LIN {X 121.514,Y -7.144,Z -55.406,A -90.000,B 90.000,C 0.000} C_DIS
LIN {X 120.744,Y -7.144,Z -56.976,A -90.000,B 90.000,C 0.000} C_DIS
LIN {X 120.185,Y -7.144,Z -58.438,A -90.000,B 90.000,C 0.000} C_DIS
LIN {X 119.652,Y -7.144,Z -59.909,A -90.000,B 90.000,C 0.000} C_DIS
LIN {X 119.147,Y -7.144,Z -61.390,A -90.000,B 90.000,C 0.000} C_DIS
LIN {X 144.015,Y -7.144,Z -61.390,A -90.000,B 90.000,C 0.000} C_DIS
LIN {X 144.015,Y -7.144,Z -68.939,A -90.000,B 90.000,C 0.000} C_DIS
LIN {X 116.917,Y -7.144,Z -68.939,A -90.000,B 90.000,C 0.000} C_DIS
LIN {X 116.287,Y -7.144,Z -70.857,A -90.000,B 90.000,C 0.000} C_DIS
LIN {X 115.601,Y -7.144,Z -72.756,A -90.000,B 90.000,C 0.000} C_DIS
LIN {X 114.859,Y -7.144,Z -74.633,A -90.000,B 90.000,C 0.000} C_DIS
LIN {X 114.062,Y -7.144,Z -76.488,A -90.000,B 90.000,C 0.000} C_DIS
LIN {X 144.015,Y -7.144,Z -76.488,A -90.000,B 90.000,C 0.000} C_DIS
LIN {X 144.015,Y -7.144,Z -84.037,A -90.000,B 90.000,C 0.000} C_DIS
LIN {X 110.374,Y -7.144,Z -84.037,A -90.000,B 90.000,C 0.000} C_DIS
LIN {X 110.982,Y -7.144,Z -85.267,A -90.000,B 90.000,C 0.000} C_DIS
LIN {X 111.542,Y -7.144,Z -86.519,A -90.000,B 90.000,C 0.000} C_DIS
LIN {X 112.054,Y -7.144,Z -87.792,A -90.000,B 90.000,C 0.000} C_DIS
LIN {X 112.517,Y -7.144,Z -89.084,A -90.000,B 90.000,C 0.000} C_DIS
LIN {X 112.888,Y -7.144,Z -90.333,A -90.000,B 90.000,C 0.000} C_DIS
LIN {X 113.248,Y -7.144,Z -91.586,A -90.000,B 90.000,C 0.000} C_DIS
LIN {X 144.015,Y -7.144,Z -91.586,A -90.000,B 90.000,C 0.000} C_DIS
LIN {X 144.015,Y -7.144,Z -99.134,A -90.000,B 90.000,C 0.000} C_DIS
LIN {X 115.197,Y -7.144,Z -99.134,A -90.000,B 90.000,C 0.000} C_DIS
LIN {X 115.413,Y -7.144,Z -100.073,A -90.000,B 90.000,C 0.000} C_DIS
LIN {X 115.939,Y -7.144,Z -102.270,A -90.000,B 90.000,C 0.000} C_DIS
LIN {X 116.438,Y -7.144,Z -104.473,A -90.000,B 90.000,C 0.000} C_DIS
LIN {X 116.908,Y -7.144,Z -106.683,A -90.000,B 90.000,C 0.000} C_DIS
LIN {X 144.015,Y -7.144,Z -106.683,A -90.000,B 90.000,C 0.000} C_DIS
LIN {X 144.015,Y -7.144,Z -114.232,A -90.000,B 90.000,C 0.000} C_DIS
LIN {X 118.297,Y -7.144,Z -114.232,A -90.000,B 90.000,C 0.000} C_DIS
LIN {X 118.685,Y -7.144,Z -116.743,A -90.000,B 90.000,C 0.000} C_DIS
LIN {X 119.037,Y -7.144,Z -119.260,A -90.000,B 90.000,C 0.000} C_DIS
LIN {X 119.354,Y -7.144,Z -121.781,A -90.000,B 90.000,C 0.000} C_DIS
LIN {X 144.015,Y -7.144,Z -121.781,A -90.000,B 90.000,C 0.000} C_DIS
LIN {X 144.015,Y -7.144,Z -129.329,A -90.000,B 90.000,C 0.000} C_DIS
LIN {X 120.084,Y -7.144,Z -129.329,A -90.000,B 90.000,C 0.000} C_DIS
LIN {X 120.256,Y -7.144,Z -131.843,A -90.000,B 90.000,C 0.000} C_DIS
LIN {X 120.392,Y -7.144,Z -134.360,A -90.000,B 90.000,C 0.000} C_DIS
LIN {X 120.492,Y -7.144,Z -136.878,A -90.000,B 90.000,C 0.000} C_DIS
LIN {X 144.015,Y -7.144,Z -136.878,A -90.000,B 90.000,C 0.000} C_DIS
LIN {X 144.015,Y -7.144,Z -144.427,A -90.000,B 90.000,C 0.000} C_DIS
LIN {X 120.524,Y -7.144,Z -144.427,A -90.000,B 90.000,C 0.000} C_DIS
LIN {X 120.468,Y -7.144,Z -148.202,A -90.000,B 90.000,C 0.000} C_DIS
LIN {X 120.375,Y -7.144,Z -151.976,A -90.000,B 90.000,C 0.000} C_DIS
LIN {X 144.015,Y -7.144,Z -151.976,A -90.000,B 90.000,C 0.000} C_DIS
LIN {X 144.015,Y -7.144,Z -159.525,A -90.000,B 90.000,C 0.000} C_DIS
LIN {X 120.081,Y -7.144,Z -159.525,A -90.000,B 90.000,C 0.000} C_DIS
LIN {X 119.879,Y -7.144,Z -163.300,A -90.000,B 90.000,C 0.000} C_DIS
LIN {X 119.641,Y -7.144,Z -167.073,A -90.000,B 90.000,C 0.000} C_DIS
LIN {X 144.015,Y -7.144,Z -167.073,A -90.000,B 90.000,C 0.000} C_DIS
LIN {X 144.015,Y -7.144,Z -174.622,A -90.000,B 90.000,C 0.000} C_DIS
LIN {X 119.054,Y -7.144,Z -174.622,A -90.000,B 90.000,C 0.000} C_DIS
LIN {X 118.705,Y -7.144,Z -178.398,A -90.000,B 90.000,C 0.000} C_DIS
LIN {X 118.321,Y -7.144,Z -182.171,A -90.000,B 90.000,C 0.000} C_DIS
LIN {X 144.015,Y -7.144,Z -182.171,A -90.000,B 90.000,C 0.000} C_DIS
LIN {X 144.015,Y -7.144,Z -189.720,A -90.000,B 90.000,C 0.000} C_DIS
LIN {X 117.439,Y -7.144,Z -189.720,A -90.000,B 90.000,C 0.000} C_DIS
LIN {X 116.942,Y -7.144,Z -193.497,A -90.000,B 90.000,C 0.000} C_DIS
LIN {X 116.409,Y -7.144,Z -197.269,A -90.000,B 90.000,C 0.000} C_DIS
LIN {X 144.015,Y -7.144,Z -197.269,A -90.000,B 90.000,C 0.000} C_DIS
LIN {X 144.015,Y -7.144,Z -204.817,A -90.000,B 90.000,C 0.000} C_DIS
LIN {X 115.297,Y -7.144,Z -204.817,A -90.000,B 90.000,C 0.000} C_DIS
LIN {X 114.880,Y -7.144,Z -207.339,A -90.000,B 90.000,C 0.000} C_DIS
LIN {X 114.433,Y -7.144,Z -209.855,A -90.000,B 90.000,C 0.000} C_DIS
LIN {X 113.956,Y -7.144,Z -212.366,A -90.000,B 90.000,C 0.000} C_DIS
LIN {X 144.015,Y -7.144,Z -212.366,A -90.000,B 90.000,C 0.000} C_DIS
LIN {X 144.015,Y -7.144,Z -219.915,A -90.000,B 90.000,C 0.000} C_DIS
LIN {X 112.335,Y -7.144,Z -219.915,A -90.000,B 90.000,C 0.000} C_DIS
LIN {X 111.729,Y -7.144,Z -222.439,A -90.000,B 90.000,C 0.000} C_DIS
LIN {X 111.093,Y -7.144,Z -224.955,A -90.000,B 90.000,C 0.000} C_DIS
LIN {X 110.426,Y -7.144,Z -227.464,A -90.000,B 90.000,C 0.000} C_DIS
LIN {X 144.015,Y -7.144,Z -227.464,A -90.000,B 90.000,C 0.000} C_DIS
LIN {X 144.015,Y -7.144,Z -235.012,A -90.000,B 90.000,C 0.000} C_DIS
LIN {X 108.222,Y -7.144,Z -235.012,A -90.000,B 90.000,C 0.000} C_DIS
LIN {X 107.417,Y -7.144,Z -237.539,A -90.000,B 90.000,C 0.000} C_DIS
LIN {X 106.580,Y -7.144,Z -240.055,A -90.000,B 90.000,C 0.000} C_DIS
LIN {X 105.713,Y -7.144,Z -242.561,A -90.000,B 90.000,C 0.000} C_DIS
LIN {X 144.015,Y -7.144,Z -242.561,A -90.000,B 90.000,C 0.000} C_DIS
LIN {X 145.015,Y -7.144,Z -243.561,A -90.000,B 90.000,C 0.000} C_DIS
LIN {X 145.015,Y -7.144,Z 0.000,A -90.000,B 90.000,C 0.000} C_DIS
LIN {X -145.015,Y -7.144,Z 0.000,A -90.000,B 90.000,C 0.000} C_DIS
LIN {X -145.015,Y -7.144,Z -243.561,A -90.000,B 90.000,C 0.000} C_DIS
LIN {X -140.554,Y -7.144,Z -243.561,A -90.000,B 90.000,C 0.000} C_DIS
LIN {X -140.119,Y -7.144,Z -242.863,A -90.000,B 90.000,C 0.000} C_DIS
LIN {X -139.634,Y -7.144,Z -242.200,A -90.000,B 90.000,C 0.000} C_DIS
LIN {X -139.100,Y -7.144,Z -241.575,A -90.000,B 90.000,C 0.000} C_DIS
LIN {X -138.520,Y -7.144,Z -240.992,A -90.000,B 90.000,C 0.000} C_DIS
LIN {X -137.899,Y -7.144,Z -240.454,A -90.000,B 90.000,C 0.000} C_DIS
LIN {X -135.929,Y -7.144,Z -239.077,A -90.000,B 90.000,C 0.000} C_DIS
LIN {X -133.939,Y -7.144,Z -237.729,A -90.000,B 90.000,C 0.000} C_DIS
LIN {X -131.929,Y -7.144,Z -236.410,A -90.000,B 90.000,C 0.000} C_DIS
LIN {X -129.901,Y -7.144,Z -235.120,A -90.000,B 90.000,C 0.000} C_DIS
LIN {X -115.273,Y -7.144,Z -225.519,A -90.000,B 90.000,C 0.000} C_DIS
LIN {X -110.220,Y -7.144,Z -222.219,A -90.000,B 90.000,C 0.000} C_DIS
LIN {X -105.138,Y -7.144,Z -218.966,A -90.000,B 90.000,C 0.000} C_DIS
LIN {X -100.026,Y -7.144,Z -215.758,A -90.000,B 90.000,C 0.000} C_DIS
LIN {X -94.885,Y -7.144,Z -212.598,A -90.000,B 90.000,C 0.000} C_DIS
LIN {X -89.715,Y -7.144,Z -209.484,A -90.000,B 90.000,C 0.000} C_DIS
LIN {X -84.517,Y -7.144,Z -206.418,A -90.000,B 90.000,C 0.000} C_DIS
LIN {X -79.291,Y -7.144,Z -203.400,A -90.000,B 90.000,C 0.000} C_DIS
LIN {X -74.039,Y -7.144,Z -200.428,A -90.000,B 90.000,C 0.000} C_DIS
LIN {X -69.832,Y -7.144,Z -198.105,A -90.000,B 90.000,C 0.000} C_DIS
LIN {X -65.646,Y -7.144,Z -195.743,A -90.000,B 90.000,C 0.000} C_DIS
LIN {X -61.483,Y -7.144,Z -193.343,A -90.000,B 90.000,C 0.000} C_DIS
LIN {X -57.342,Y -7.144,Z -190.904,A -90.000,B 90.000,C 0.000} C_DIS
LIN {X -53.223,Y -7.144,Z -188.427,A -90.000,B 90.000,C 0.000} C_DIS
LIN {X -50.631,Y -7.144,Z -186.839,A -90.000,B 90.000,C 0.000} C_DIS
LIN {X -48.069,Y -7.144,Z -185.203,A -90.000,B 90.000,C 0.000} C_DIS
LIN {X -45.539,Y -7.144,Z -183.518,A -90.000,B 90.000,C 0.000} C_DIS
LIN {X -43.042,Y -7.144,Z -181.785,A -90.000,B 90.000,C 0.000} C_DIS
LIN {X -40.578,Y -7.144,Z -180.005,A -90.000,B 90.000,C 0.000} C_DIS
LIN {X -38.149,Y -7.144,Z -178.178,A -90.000,B 90.000,C 0.000} C_DIS
LIN {X -35.754,Y -7.144,Z -176.305,A -90.000,B 90.000,C 0.000} C_DIS
LIN {X -33.396,Y -7.144,Z -174.387,A -90.000,B 90.000,C 0.000} C_DIS
LIN {X -32.331,Y -7.144,Z -173.515,A -90.000,B 90.000,C 0.000} C_DIS
LIN {X -31.313,Y -7.144,Z -172.588,A -90.000,B 90.000,C 0.000} C_DIS
LIN {X -30.343,Y -7.144,Z -171.611,A -90.000,B 90.000,C 0.000} C_DIS
LIN {X -29.426,Y -7.144,Z -170.585,A -90.000,B 90.000,C 0.000} C_DIS
LIN {X -28.562,Y -7.144,Z -169.513,A -90.000,B 90.000,C 0.000} C_DIS
LIN {X -27.755,Y -7.144,Z -168.398,A -90.000,B 90.000,C 0.000} C_DIS
LIN {X -27.006,Y -7.144,Z -167.243,A -90.000,B 90.000,C 0.000} C_DIS
LIN {X -26.318,Y -7.144,Z -166.051,A -90.000,B 90.000,C 0.000} C_DIS
LIN {X -25.692,Y -7.144,Z -164.825,A -90.000,B 90.000,C 0.000} C_DIS
LIN {X -25.130,Y -7.144,Z -163.568,A -90.000,B 90.000,C 0.000} C_DIS
LIN {X -24.634,Y -7.144,Z -162.284,A -90.000,B 90.000,C 0.000} C_DIS
LIN {X -24.737,Y -7.144,Z -162.088,A -90.000,B 90.000,C 0.000} C_DIS
LIN {X -25.690,Y -7.144,Z -160.813,A -90.000,B 90.000,C 0.000} C_DIS
LIN {X -26.684,Y -7.144,Z -159.569,A -90.000,B 90.000,C 0.000} C_DIS
LIN {X -27.716,Y -7.144,Z -158.357,A -90.000,B 90.000,C 0.000} C_DIS
LIN {X -28.785,Y -7.144,Z -157.178,A -90.000,B 90.000,C 0.000} C_DIS
LIN {X -29.891,Y -7.144,Z -156.033,A -90.000,B 90.000,C 0.000} C_DIS
LIN {X -31.033,Y -7.144,Z -154.924,A -90.000,B 90.000,C 0.000} C_DIS
LIN {X -32.331,Y -7.144,Z -153.550,A -90.000,B 90.000,C 0.000} C_DIS
LIN {X -33.595,Y -7.144,Z -152.143,A -90.000,B 90.000,C 0.000} C_DIS
LIN {X -34.822,Y -7.144,Z -150.705,A -90.000,B 90.000,C 0.000} C_DIS
LIN {X -36.012,Y -7.144,Z -149.236,A -90.000,B 90.000,C 0.000} C_DIS
LIN {X -37.165,Y -7.144,Z -147.738,A -90.000,B 90.000,C 0.000} C_DIS
LIN {X -38.280,Y -7.144,Z -146.211,A -90.000,B 90.000,C 0.000} C_DIS
LIN {X -39.590,Y -7.144,Z -144.190,A -90.000,B 90.000,C 0.000} C_DIS
LIN {X -40.845,Y -7.144,Z -142.134,A -90.000,B 90.000,C 0.000} C_DIS
LIN {X -42.044,Y -7.144,Z -140.045,A -90.000,B 90.000,C 0.000} C_DIS
LIN {X -43.186,Y -7.144,Z -137.924,A -90.000,B 90.000,C 0.000} C_DIS
LIN {X -44.271,Y -7.144,Z -135.774,A -90.000,B 90.000,C 0.000} C_DIS
LIN {X -45.298,Y -7.144,Z -133.595,A -90.000,B 90.000,C 0.000} C_DIS
LIN {X -46.265,Y -7.144,Z -131.389,A -90.000,B 90.000,C 0.000} C_DIS
LIN {X -46.906,Y -7.144,Z -129.756,A -90.000,B 90.000,C 0.000} C_DIS
LIN {X -47.592,Y -7.144,Z -128.142,A -90.000,B 90.000,C 0.000} C_DIS
LIN {X -48.322,Y -7.144,Z -126.547,A -90.000,B 90.000,C 0.000} C_DIS
LIN {X -49.096,Y -7.144,Z -124.973,A -90.000,B 90.000,C 0.000} C_DIS
LIN {X -50.069,Y -7.144,Z -123.522,A -90.000,B 90.000,C 0.000} C_DIS
LIN {X -51.086,Y -7.144,Z -122.102,A -90.000,B 90.000,C 0.000} C_DIS
LIN {X -52.147,Y -7.144,Z -120.715,A -90.000,B 90.000,C 0.000} C_DIS
LIN {X -53.250,Y -7.144,Z -119.360,A -90.000,B 90.000,C 0.000} C_DIS
LIN {X -55.412,Y -7.144,Z -116.608,A -90.000,B 90.000,C 0.000} C_DIS
LIN {X -57.611,Y -7.144,Z -113.887,A -90.000,B 90.000,C 0.000} C_DIS
LIN {X -59.849,Y -7.144,Z -111.197,A -90.000,B 90.000,C 0.000} C_DIS
LIN {X -62.123,Y -7.144,Z -108.538,A -90.000,B 90.000,C 0.000} C_DIS
LIN {X -64.435,Y -7.144,Z -105.911,A -90.000,B 90.000,C 0.000} C_DIS
LIN {X -65.822,Y -7.144,Z -104.451,A -90.000,B 90.000,C 0.000} C_DIS
LIN {X -67.253,Y -7.144,Z -103.034,A -90.000,B 90.000,C 0.000} C_DIS
LIN {X -68.726,Y -7.144,Z -101.661,A -90.000,B 90.000,C 0.000} C_DIS
LIN {X -70.240,Y -7.144,Z -100.334,A -90.000,B 90.000,C 0.000} C_DIS
LIN {X -71.793,Y -7.144,Z -99.053,A -90.000,B 90.000,C 0.000} C_DIS
LIN {X -73.385,Y -7.144,Z -97.819,A -90.000,B 90.000,C 0.000} C_DIS
LIN {X -75.013,Y -7.144,Z -96.634,A -90.000,B 90.000,C 0.000} C_DIS
LIN {X -76.677,Y -7.144,Z -95.500,A -90.000,B 90.000,C 0.000} C_DIS
LIN {X -78.374,Y -7.144,Z -94.416,A -90.000,B 90.000,C 0.000} C_DIS
LIN {X -80.315,Y -7.144,Z -93.198,A -90.000,B 90.000,C 0.000} C_DIS
LIN {X -82.246,Y -7.144,Z -91.965,A -90.000,B 90.000,C 0.000} C_DIS
LIN {X -85.301,Y -7.144,Z -89.688,A -90.000,B 90.000,C 0.000} C_DIS
LIN {X -88.370,Y -7.144,Z -87.432,A -90.000,B 90.000,C 0.000} C_DIS
LIN {X -90.228,Y -7.144,Z -86.171,A -90.000,B 90.000,C 0.000} C_DIS
LIN {X -92.071,Y -7.144,Z -84.889,A -90.000,B 90.000,C 0.000} C_DIS
LIN {X -93.338,Y -7.144,Z -84.976,A -90.000,B 90.000,C 0.000} C_DIS
LIN {X -94.608,Y -7.144,Z -84.998,A -90.000,B 90.000,C 0.000} C_DIS
LIN {X -95.877,Y -7.144,Z -84.956,A -90.000,B 90.000,C 0.000} C_DIS
LIN {X -97.143,Y -7.144,Z -84.850,A -90.000,B 90.000,C 0.000} C_DIS
LIN {X -98.401,Y -7.144,Z -84.679,A -90.000,B 90.000,C 0.000} C_DIS
LIN {X -99.650,Y -7.144,Z -84.445,A -90.000,B 90.000,C 0.000} C_DIS
LIN {X -100.884,Y -7.144,Z -84.148,A -90.000,B 90.000,C 0.000} C_DIS
LIN {X -102.103,Y -7.144,Z -83.788,A -90.000,B 90.000,C 0.000} C_DIS
LIN {X -103.301,Y -7.144,Z -83.368,A -90.000,B 90.000,C 0.000} C_DIS
LIN {X -104.689,Y -7.144,Z -82.711,A -90.000,B 90.000,C 0.000} C_DIS
LIN {X -106.045,Y -7.144,Z -81.991,A -90.000,B 90.000,C 0.000} C_DIS
LIN {X -107.368,Y -7.144,Z -81.211,A -90.000,B 90.000,C 0.000} C_DIS
LIN {X -108.654,Y -7.144,Z -80.372,A -90.000,B 90.000,C 0.000} C_DIS
LIN {X -109.900,Y -7.144,Z -79.475,A -90.000,B 90.000,C 0.000} C_DIS
LIN {X -111.105,Y -7.144,Z -78.523,A -90.000,B 90.000,C 0.000} C_DIS
LIN {X -112.265,Y -7.144,Z -77.517,A -90.000,B 90.000,C 0.000} C_DIS
LIN {X -113.379,Y -7.144,Z -76.460,A -90.000,B 90.000,C 0.000} C_DIS
LIN {X -114.443,Y -7.144,Z -75.354,A -90.000,B 90.000,C 0.000} C_DIS
LIN {X -115.456,Y -7.144,Z -74.200,A -90.000,B 90.000,C 0.000} C_DIS
LIN {X -116.417,Y -7.144,Z -73.002,A -90.000,B 90.000,C 0.000} C_DIS
LIN {X -117.321,Y -7.144,Z -71.761,A -90.000,B 90.000,C 0.000} C_DIS
LIN {X -118.114,Y -7.144,Z -70.320,A -90.000,B 90.000,C 0.000} C_DIS
LIN {X -118.859,Y -7.144,Z -68.854,A -90.000,B 90.000,C 0.000} C_DIS
LIN {X -119.555,Y -7.144,Z -67.364,A -90.000,B 90.000,C 0.000} C_DIS
LIN {X -120.202,Y -7.144,Z -65.852,A -90.000,B 90.000,C 0.000} C_DIS
LIN {X -120.798,Y -7.144,Z -64.319,A -90.000,B 90.000,C 0.000} C_DIS
LIN {X -121.344,Y -7.144,Z -62.768,A -90.000,B 90.000,C 0.000} C_DIS
LIN {X -121.997,Y -7.144,Z -60.822,A -90.000,B 90.000,C 0.000} C_DIS
LIN {X -122.664,Y -7.144,Z -58.882,A -90.000,B 90.000,C 0.000} C_DIS
LIN {X -123.168,Y -7.144,Z -57.739,A -90.000,B 90.000,C 0.000} C_DIS
LIN {X -123.625,Y -7.144,Z -56.577,A -90.000,B 90.000,C 0.000} C_DIS
LIN {X -124.036,Y -7.144,Z -55.398,A -90.000,B 90.000,C 0.000} C_DIS
LIN {X -124.398,Y -7.144,Z -54.203,A -90.000,B 90.000,C 0.000} C_DIS
LIN {X -124.712,Y -7.144,Z -52.994,A -90.000,B 90.000,C 0.000} C_DIS
LIN {X -124.968,Y -7.144,Z -52.047,A -90.000,B 90.000,C 0.000} C_DIS
LIN {X -125.160,Y -7.144,Z -51.085,A -90.000,B 90.000,C 0.000} C_DIS
LIN {X -125.286,Y -7.144,Z -50.113,A -90.000,B 90.000,C 0.000} C_DIS
LIN {X -125.346,Y -7.144,Z -49.134,A -90.000,B 90.000,C 0.000} C_DIS
LIN {X -125.339,Y -7.144,Z -48.153,A -90.000,B 90.000,C 0.000} C_DIS
LIN {X -125.267,Y -7.144,Z -47.175,A -90.000,B 90.000,C 0.000} C_DIS
LIN {X -125.128,Y -7.144,Z -46.204,A -90.000,B 90.000,C 0.000} C_DIS
LIN {X -125.580,Y -7.144,Z -44.284,A -90.000,B 90.000,C 0.000} C_DIS
LIN {X -125.752,Y -7.144,Z -43.367,A -90.000,B 90.000,C 0.000} C_DIS
LIN {X -125.861,Y -7.144,Z -42.440,A -90.000,B 90.000,C 0.000} C_DIS
LIN {X -125.905,Y -7.144,Z -41.508,A -90.000,B 90.000,C 0.000} C_DIS
LIN {X -125.885,Y -7.144,Z -40.575,A -90.000,B 90.000,C 0.000} C_DIS
LIN {X -125.801,Y -7.144,Z -39.645,A -90.000,B 90.000,C 0.000} C_DIS
LIN {X -125.652,Y -7.144,Z -38.724,A -90.000,B 90.000,C 0.000} C_DIS
LIN {X -125.441,Y -7.144,Z -37.815,A -90.000,B 90.000,C 0.000} C_DIS
LIN {X -125.167,Y -7.144,Z -36.923,A -90.000,B 90.000,C 0.000} C_DIS
LIN {X -125.301,Y -7.144,Z -35.857,A -90.000,B 90.000,C 0.000} C_DIS
LIN {X -125.366,Y -7.144,Z -34.784,A -90.000,B 90.000,C 0.000} C_DIS
LIN {X -125.361,Y -7.144,Z -33.710,A -90.000,B 90.000,C 0.000} C_DIS
LIN {X -125.286,Y -7.144,Z -32.638,A -90.000,B 90.000,C 0.000} C_DIS
LIN {X -125.142,Y -7.144,Z -31.573,A -90.000,B 90.000,C 0.000} C_DIS
LIN {X -124.929,Y -7.144,Z -30.520,A -90.000,B 90.000,C 0.000} C_DIS
LIN {X -124.648,Y -7.144,Z -29.483,A -90.000,B 90.000,C 0.000} C_DIS
LIN {X -124.300,Y -7.144,Z -28.467,A -90.000,B 90.000,C 0.000} C_DIS
LIN {X -123.887,Y -7.144,Z -27.475,A -90.000,B 90.000,C 0.000} C_DIS
LIN {X -123.410,Y -7.144,Z -26.512,A -90.000,B 90.000,C 0.000} C_DIS
LIN {X -122.871,Y -7.144,Z -25.582,A -90.000,B 90.000,C 0.000} C_DIS
LIN {X -122.274,Y -7.144,Z -24.689,A -90.000,B 90.000,C 0.000} C_DIS
LIN {X -121.619,Y -7.144,Z -23.837,A -90.000,B 90.000,C 0.000} C_DIS
LIN {X -120.911,Y -7.144,Z -23.029,A -90.000,B 90.000,C 0.000} C_DIS
LIN {X -120.459,Y -7.144,Z -22.157,A -90.000,B 90.000,C 0.000} C_DIS
LIN {X -119.954,Y -7.144,Z -21.315,A -90.000,B 90.000,C 0.000} C_DIS
LIN {X -119.400,Y -7.144,Z -20.504,A -90.000,B 90.000,C 0.000} C_DIS
LIN {X -118.797,Y -7.144,Z -19.729,A -90.000,B 90.000,C 0.000} C_DIS
LIN {X -118.148,Y -7.144,Z -18.992,A -90.000,B 90.000,C 0.000} C_DIS
LIN {X -117.455,Y -7.144,Z -18.296,A -90.000,B 90.000,C 0.000} C_DIS
LIN {X -116.519,Y -7.144,Z -17.499,A -90.000,B 90.000,C 0.000} C_DIS
LIN {X -115.538,Y -7.144,Z -16.758,A -90.000,B 90.000,C 0.000} C_DIS
LIN {X -114.517,Y -7.144,Z -16.074,A -90.000,B 90.000,C 0.000} C_DIS
LIN {X -113.457,Y -7.144,Z -15.451,A -90.000,B 90.000,C 0.000} C_DIS
LIN {X -112.364,Y -7.144,Z -14.889,A -90.000,B 90.000,C 0.000} C_DIS
LIN {X -111.240,Y -7.144,Z -14.391,A -90.000,B 90.000,C 0.000} C_DIS
LIN {X -110.089,Y -7.144,Z -13.959,A -90.000,B 90.000,C 0.000} C_DIS
LIN {X -108.915,Y -7.144,Z -13.594,A -90.000,B 90.000,C 0.000} C_DIS
LIN {X -107.722,Y -7.144,Z -13.298,A -90.000,B 90.000,C 0.000} C_DIS
LIN {X -106.514,Y -7.144,Z -13.070,A -90.000,B 90.000,C 0.000} C_DIS
LIN {X -105.295,Y -7.144,Z -12.913,A -90.000,B 90.000,C 0.000} C_DIS
LIN {X -104.195,Y -7.144,Z -12.093,A -90.000,B 90.000,C 0.000} C_DIS
LIN {X -102.641,Y -7.144,Z -11.193,A -90.000,B 90.000,C 0.000} C_DIS
LIN {X -101.059,Y -7.144,Z -10.343,A -90.000,B 90.000,C 0.000} C_DIS
LIN {X -99.452,Y -7.144,Z -9.543,A -90.000,B 90.000,C 0.000} C_DIS
LIN {X -97.820,Y -7.144,Z -8.793,A -90.000,B 90.000,C 0.000} C_DIS
LIN {X -96.165,Y -7.144,Z -8.096,A -90.000,B 90.000,C 0.000} C_DIS
LIN {X -94.489,Y -7.144,Z -7.451,A -90.000,B 90.000,C 0.000} C_DIS
LIN {X -92.683,Y -7.144,Z -6.908,A -90.000,B 90.000,C 0.000} C_DIS
LIN {X -90.861,Y -7.144,Z -6.427,A -90.000,B 90.000,C 0.000} C_DIS
LIN {X -89.023,Y -7.144,Z -6.006,A -90.000,B 90.000,C 0.000} C_DIS
LIN {X -87.172,Y -7.144,Z -5.648,A -90.000,B 90.000,C 0.000} C_DIS
LIN {X -85.310,Y -7.144,Z -5.352,A -90.000,B 90.000,C 0.000} C_DIS
LIN {X -83.439,Y -7.144,Z -5.119,A -90.000,B 90.000,C 0.000} C_DIS
LIN {X -81.561,Y -7.144,Z -4.949,A -90.000,B 90.000,C 0.000} C_DIS
LIN {X -79.679,Y -7.144,Z -4.842,A -90.000,B 90.000,C 0.000} C_DIS
LIN {X -77.794,Y -7.144,Z -4.799,A -90.000,B 90.000,C 0.000} C_DIS
LIN {X -75.909,Y -7.144,Z -4.818,A -90.000,B 90.000,C 0.000} C_DIS
LIN {X -74.025,Y -7.144,Z -4.901,A -90.000,B 90.000,C 0.000} C_DIS
LIN {X -72.146,Y -7.144,Z -5.048,A -90.000,B 90.000,C 0.000} C_DIS
LIN {X -70.272,Y -7.144,Z -5.257,A -90.000,B 90.000,C 0.000} C_DIS
LIN {X -68.578,Y -7.144,Z -5.307,A -90.000,B 90.000,C 0.000} C_DIS
LIN {X -66.884,Y -7.144,Z -5.392,A -90.000,B 90.000,C 0.000} C_DIS
LIN {X -65.193,Y -7.144,Z -5.511,A -90.000,B 90.000,C 0.000} C_DIS
LIN {X -63.505,Y -7.144,Z -5.664,A -90.000,B 90.000,C 0.000} C_DIS
LIN {X -61.132,Y -7.144,Z -6.143,A -90.000,B 90.000,C 0.000} C_DIS
LIN {X -58.771,Y -7.144,Z -6.678,A -90.000,B 90.000,C 0.000} C_DIS
LIN {X -56.424,Y -7.144,Z -7.268,A -90.000,B 90.000,C 0.000} C_DIS
LIN {X -54.091,Y -7.144,Z -7.914,A -90.000,B 90.000,C 0.000} C_DIS
LIN {X -52.131,Y -7.144,Z -8.508,A -90.000,B 90.000,C 0.000} C_DIS
LIN {X -50.156,Y -7.144,Z -9.051,A -90.000,B 90.000,C 0.000} C_DIS
LIN {X -48.168,Y -7.144,Z -9.544,A -90.000,B 90.000,C 0.000} C_DIS
LIN {X -46.169,Y -7.144,Z -9.985,A -90.000,B 90.000,C 0.000} C_DIS
LIN {X -44.158,Y -7.144,Z -10.375,A -90.000,B 90.000,C 0.000} C_DIS
LIN {X -39.354,Y -7.144,Z -11.215,A -90.000,B 90.000,C 0.000} C_DIS
LIN {X -34.561,Y -7.144,Z -12.113,A -90.000,B 90.000,C 0.000} C_DIS
LIN {X -29.780,Y -7.144,Z -13.070,A -90.000,B 90.000,C 0.000} C_DIS
LIN {X -25.011,Y -7.144,Z -14.086,A -90.000,B 90.000,C 0.000} C_DIS
LIN {X -20.254,Y -7.144,Z -15.161,A -90.000,B 90.000,C 0.000} C_DIS
LIN {X -15.511,Y -7.144,Z -16.294,A -90.000,B 90.000,C 0.000} C_DIS
LIN {X -10.451,Y -7.144,Z -17.735,A -90.000,B 90.000,C 0.000} C_DIS
LIN {X -5.383,Y -7.144,Z -19.147,A -90.000,B 90.000,C 0.000} C_DIS
LIN {X -0.306,Y -7.144,Z -20.529,A -90.000,B 90.000,C 0.000} C_DIS
LIN {X 4.586,Y -7.144,Z -21.651,A -90.000,B 90.000,C 0.000} C_DIS
LIN {X 9.469,Y -7.144,Z -22.811,A -90.000,B 90.000,C 0.000} C_DIS
LIN {X 14.343,Y -7.144,Z -24.010,A -90.000,B 90.000,C 0.000} C_DIS
LIN {X 17.619,Y -7.144,Z -24.747,A -90.000,B 90.000,C 0.000} C_DIS
LIN {X 20.887,Y -7.144,Z -25.514,A -90.000,B 90.000,C 0.000} C_DIS
LIN {X 23.040,Y -7.144,Z -25.870,A -90.000,B 90.000,C 0.000} C_DIS
LIN {X 25.182,Y -7.144,Z -26.288,A -90.000,B 90.000,C 0.000} C_DIS
LIN {X 27.311,Y -7.144,Z -26.766,A -90.000,B 90.000,C 0.000} C_DIS
LIN {X 29.426,Y -7.144,Z -27.305,A -90.000,B 90.000,C 0.000} C_DIS
LIN {X 31.524,Y -7.144,Z -27.904,A -90.000,B 90.000,C 0.000} C_DIS
LIN {X 33.605,Y -7.144,Z -28.561,A -90.000,B 90.000,C 0.000} C_DIS
LIN {X 37.148,Y -7.144,Z -29.729,A -90.000,B 90.000,C 0.000} C_DIS
LIN {X 40.701,Y -7.144,Z -30.867,A -90.000,B 90.000,C 0.000} C_DIS
LIN {X 43.526,Y -7.144,Z -31.707,A -90.000,B 90.000,C 0.000} C_DIS
LIN {X 46.333,Y -7.144,Z -32.607,A -90.000,B 90.000,C 0.000} C_DIS
LIN {X 49.119,Y -7.144,Z -33.567,A -90.000,B 90.000,C 0.000} C_DIS
LIN {X 51.885,Y -7.144,Z -34.587,A -90.000,B 90.000,C 0.000} C_DIS
LIN {X 54.627,Y -7.144,Z -35.666,A -90.000,B 90.000,C 0.000} C_DIS
LIN {X 57.346,Y -7.144,Z -36.804,A -90.000,B 90.000,C 0.000} C_DIS
LIN {X 60.037,Y -7.144,Z -38.079,A -90.000,B 90.000,C 0.000} C_DIS
LIN {X 62.703,Y -7.144,Z -39.406,A -90.000,B 90.000,C 0.000} C_DIS
LIN {X 65.342,Y -7.144,Z -40.785,A -90.000,B 90.000,C 0.000} C_DIS
LIN {X 67.954,Y -7.144,Z -42.216,A -90.000,B 90.000,C 0.000} C_DIS
LIN {X 70.537,Y -7.144,Z -43.698,A -90.000,B 90.000,C 0.000} C_DIS
LIN {X 73.090,Y -7.144,Z -45.230,A -90.000,B 90.000,C 0.000} C_DIS
LIN {X 75.613,Y -7.144,Z -46.812,A -90.000,B 90.000,C 0.000} C_DIS
LIN {X 78.105,Y -7.144,Z -48.443,A -90.000,B 90.000,C 0.000} C_DIS
LIN {X 79.011,Y -7.144,Z -47.146,A -90.000,B 90.000,C 0.000} C_DIS
LIN {X 79.967,Y -7.144,Z -45.887,A -90.000,B 90.000,C 0.000} C_DIS
LIN {X 80.973,Y -7.144,Z -44.666,A -90.000,B 90.000,C 0.000} C_DIS
LIN {X 82.026,Y -7.144,Z -43.486,A -90.000,B 90.000,C 0.000} C_DIS
LIN {X 83.125,Y -7.144,Z -42.348,A -90.000,B 90.000,C 0.000} C_DIS
LIN {X 84.268,Y -7.144,Z -41.255,A -90.000,B 90.000,C 0.000} C_DIS
LIN {X 85.454,Y -7.144,Z -40.208,A -90.000,B 90.000,C 0.000} C_DIS
LIN {X 86.680,Y -7.144,Z -39.209,A -90.000,B 90.000,C 0.000} C_DIS
LIN {X 87.945,Y -7.144,Z -38.259,A -90.000,B 90.000,C 0.000} C_DIS
LIN {X 89.246,Y -7.144,Z -37.360,A -90.000,B 90.000,C 0.000} C_DIS
LIN {X 91.067,Y -7.144,Z -36.216,A -90.000,B 90.000,C 0.000} C_DIS
LIN {X 92.918,Y -7.144,Z -35.121,A -90.000,B 90.000,C 0.000} C_DIS
LIN {X 94.797,Y -7.144,Z -34.076,A -90.000,B 90.000,C 0.000} C_DIS
LIN {X 96.704,Y -7.144,Z -33.081,A -90.000,B 90.000,C 0.000} C_DIS
LIN {X 98.636,Y -7.144,Z -32.137,A -90.000,B 90.000,C 0.000} C_DIS
LIN {X 100.592,Y -7.144,Z -31.245,A -90.000,B 90.000,C 0.000} C_DIS
LIN {X 102.572,Y -7.144,Z -30.405,A -90.000,B 90.000,C 0.000} C_DIS
LIN {X 104.573,Y -7.144,Z -29.618,A -90.000,B 90.000,C 0.000} C_DIS
LIN {X 105.549,Y -7.144,Z -29.229,A -90.000,B 90.000,C 0.000} C_DIS
LIN {X 106.550,Y -7.144,Z -28.913,A -90.000,B 90.000,C 0.000} C_DIS
LIN {X 107.572,Y -7.144,Z -28.670,A -90.000,B 90.000,C 0.000} C_DIS
LIN {X 108.608,Y -7.144,Z -28.501,A -90.000,B 90.000,C 0.000} C_DIS
LIN {X 109.655,Y -7.144,Z -28.409,A -90.000,B 90.000,C 0.000} C_DIS
LIN {X 110.705,Y -7.144,Z -28.392,A -90.000,B 90.000,C 0.000} C_DIS
LIN {X 111.753,Y -7.144,Z -28.452,A -90.000,B 90.000,C 0.000} C_DIS
LIN {X 112.795,Y -7.144,Z -28.588,A -90.000,B 90.000,C 0.000} C_DIS
LIN {X 113.824,Y -7.144,Z -28.800,A -90.000,B 90.000,C 0.000} C_DIS
LIN {X 114.834,Y -7.144,Z -29.085,A -90.000,B 90.000,C 0.000} C_DIS
LIN {X 115.822,Y -7.144,Z -29.443,A -90.000,B 90.000,C 0.000} C_DIS
LIN {X 116.780,Y -7.144,Z -29.872,A -90.000,B 90.000,C 0.000} C_DIS
LIN {X 117.705,Y -7.144,Z -30.370,A -90.000,B 90.000,C 0.000} C_DIS
LIN {X 118.592,Y -7.144,Z -30.933,A -90.000,B 90.000,C 0.000} C_DIS
LIN {X 119.435,Y -7.144,Z -31.559,A -90.000,B 90.000,C 0.000} C_DIS
LIN {X 120.230,Y -7.144,Z -32.245,A -90.000,B 90.000,C 0.000} C_DIS
LIN {X 120.974,Y -7.144,Z -32.986,A -90.000,B 90.000,C 0.000} C_DIS
LIN {X 121.662,Y -7.144,Z -33.780,A -90.000,B 90.000,C 0.000} C_DIS
LIN {X 122.196,Y -7.144,Z -34.612,A -90.000,B 90.000,C 0.000} C_DIS
LIN {X 122.676,Y -7.144,Z -35.476,A -90.000,B 90.000,C 0.000} C_DIS
LIN {X 123.102,Y -7.144,Z -36.368,A -90.000,B 90.000,C 0.000} C_DIS
LIN {X 123.470,Y -7.144,Z -37.286,A -90.000,B 90.000,C 0.000} C_DIS
LIN {X 123.781,Y -7.144,Z -38.224,A -90.000,B 90.000,C 0.000} C_DIS
LIN {X 124.032,Y -7.144,Z -39.180,A -90.000,B 90.000,C 0.000} C_DIS
LIN {X 124.222,Y -7.144,Z -40.150,A -90.000,B 90.000,C 0.000} C_DIS
LIN {X 124.352,Y -7.144,Z -41.130,A -90.000,B 90.000,C 0.000} C_DIS
LIN {X 124.419,Y -7.144,Z -42.117,A -90.000,B 90.000,C 0.000} C_DIS
LIN {X 124.425,Y -7.144,Z -43.105,A -90.000,B 90.000,C 0.000} C_DIS
LIN {X 124.369,Y -7.144,Z -44.092,A -90.000,B 90.000,C 0.000} C_DIS
LIN {X 124.170,Y -7.144,Z -45.366,A -90.000,B 90.000,C 0.000} C_DIS
LIN {X 123.911,Y -7.144,Z -46.630,A -90.000,B 90.000,C 0.000} C_DIS
LIN {X 123.595,Y -7.144,Z -47.880,A -90.000,B 90.000,C 0.000} C_DIS
LIN {X 123.220,Y -7.144,Z -49.114,A -90.000,B 90.000,C 0.000} C_DIS
LIN {X 122.789,Y -7.144,Z -50.330,A -90.000,B 90.000,C 0.000} C_DIS
LIN {X 122.302,Y -7.144,Z -51.524,A -90.000,B 90.000,C 0.000} C_DIS
LIN {X 121.760,Y -7.144,Z -52.694,A -90.000,B 90.000,C 0.000} C_DIS
LIN {X 120.784,Y -7.144,Z -54.629,A -90.000,B 90.000,C 0.000} C_DIS
LIN {X 119.828,Y -7.144,Z -56.574,A -90.000,B 90.000,C 0.000} C_DIS
LIN {X 119.134,Y -7.144,Z -58.398,A -90.000,B 90.000,C 0.000} C_DIS
LIN {X 118.481,Y -7.144,Z -60.236,A -90.000,B 90.000,C 0.000} C_DIS
LIN {X 117.869,Y -7.144,Z -62.089,A -90.000,B 90.000,C 0.000} C_DIS
LIN {X 117.300,Y -7.144,Z -63.956,A -90.000,B 90.000,C 0.000} C_DIS
LIN {X 116.772,Y -7.144,Z -65.834,A -90.000,B 90.000,C 0.000} C_DIS
LIN {X 116.180,Y -7.144,Z -67.927,A -90.000,B 90.000,C 0.000} C_DIS
LIN {X 115.522,Y -7.144,Z -70.000,A -90.000,B 90.000,C 0.000} C_DIS
LIN {X 114.797,Y -7.144,Z -72.050,A -90.000,B 90.000,C 0.000} C_DIS
LIN {X 114.006,Y -7.144,Z -74.077,A -90.000,B 90.000,C 0.000} C_DIS
LIN {X 113.150,Y -7.144,Z -76.076,A -90.000,B 90.000,C 0.000} C_DIS
LIN {X 112.230,Y -7.144,Z -78.047,A -90.000,B 90.000,C 0.000} C_DIS
LIN {X 111.248,Y -7.144,Z -79.987,A -90.000,B 90.000,C 0.000} C_DIS
LIN {X 110.203,Y -7.144,Z -81.895,A -90.000,B 90.000,C 0.000} C_DIS
LIN {X 109.097,Y -7.144,Z -83.768,A -90.000,B 90.000,C 0.000} C_DIS
LIN {X 109.669,Y -7.144,Z -84.856,A -90.000,B 90.000,C 0.000} C_DIS
LIN {X 110.203,Y -7.144,Z -85.963,A -90.000,B 90.000,C 0.000} C_DIS
LIN {X 110.697,Y -7.144,Z -87.088,A -90.000,B 90.000,C 0.000} C_DIS
LIN {X 111.151,Y -7.144,Z -88.230,A -90.000,B 90.000,C 0.000} C_DIS
LIN {X 111.564,Y -7.144,Z -89.388,A -90.000,B 90.000,C 0.000} C_DIS
LIN {X 112.354,Y -7.144,Z -92.098,A -90.000,B 90.000,C 0.000} C_DIS
LIN {X 113.096,Y -7.144,Z -94.821,A -90.000,B 90.000,C 0.000} C_DIS
LIN {X 113.792,Y -7.144,Z -97.556,A -90.000,B 90.000,C 0.000} C_DIS
LIN {X 114.440,Y -7.144,Z -100.303,A -90.000,B 90.000,C 0.000} C_DIS
LIN {X 115.248,Y -7.144,Z -103.730,A -90.000,B 90.000,C 0.000} C_DIS
LIN {X 115.988,Y -7.144,Z -107.172,A -90.000,B 90.000,C 0.000} C_DIS
LIN {X 116.659,Y -7.144,Z -110.629,A -90.000,B 90.000,C 0.000} C_DIS
LIN {X 117.262,Y -7.144,Z -114.098,A -90.000,B 90.000,C 0.000} C_DIS
LIN {X 117.796,Y -7.144,Z -117.578,A -90.000,B 90.000,C 0.000} C_DIS
LIN {X 118.260,Y -7.144,Z -121.068,A -90.000,B 90.000,C 0.000} C_DIS
LIN {X 118.655,Y -7.144,Z -124.567,A -90.000,B 90.000,C 0.000} C_DIS
LIN {X 118.981,Y -7.144,Z -128.072,A -90.000,B 90.000,C 0.000} C_DIS
LIN {X 119.237,Y -7.144,Z -131.584,A -90.000,B 90.000,C 0.000} C_DIS
LIN {X 119.424,Y -7.144,Z -135.100,A -90.000,B 90.000,C 0.000} C_DIS
LIN {X 119.540,Y -7.144,Z -138.619,A -90.000,B 90.000,C 0.000} C_DIS
LIN {X 119.531,Y -7.144,Z -143.704,A -90.000,B 90.000,C 0.000} C_DIS
LIN {X 119.456,Y -7.144,Z -148.788,A -90.000,B 90.000,C 0.000} C_DIS
LIN {X 119.314,Y -7.144,Z -153.871,A -90.000,B 90.000,C 0.000} C_DIS
LIN {X 119.107,Y -7.144,Z -158.951,A -90.000,B 90.000,C 0.000} C_DIS
LIN {X 118.834,Y -7.144,Z -164.029,A -90.000,B 90.000,C 0.000} C_DIS
LIN {X 118.494,Y -7.144,Z -169.102,A -90.000,B 90.000,C 0.000} C_DIS
LIN {X 118.089,Y -7.144,Z -174.171,A -90.000,B 90.000,C 0.000} C_DIS
LIN {X 117.618,Y -7.144,Z -179.233,A -90.000,B 90.000,C 0.000} C_DIS
LIN {X 117.082,Y -7.144,Z -184.290,A -90.000,B 90.000,C 0.000} C_DIS
LIN {X 116.479,Y -7.144,Z -189.339,A -90.000,B 90.000,C 0.000} C_DIS
LIN {X 115.811,Y -7.144,Z -194.379,A -90.000,B 90.000,C 0.000} C_DIS
LIN {X 115.078,Y -7.144,Z -199.411,A -90.000,B 90.000,C 0.000} C_DIS
LIN {X 114.541,Y -7.144,Z -203.167,A -90.000,B 90.000,C 0.000} C_DIS
LIN {X 113.938,Y -7.144,Z -206.913,A -90.000,B 90.000,C 0.000} C_DIS
LIN {X 113.268,Y -7.144,Z -210.648,A -90.000,B 90.000,C 0.000} C_DIS
LIN {X 112.532,Y -7.144,Z -214.371,A -90.000,B 90.000,C 0.000} C_DIS
LIN {X 111.730,Y -7.144,Z -218.079,A -90.000,B 90.000,C 0.000} C_DIS
LIN {X 110.862,Y -7.144,Z -221.773,A -90.000,B 90.000,C 0.000} C_DIS
LIN {X 109.929,Y -7.144,Z -225.451,A -90.000,B 90.000,C 0.000} C_DIS
LIN {X 108.931,Y -7.144,Z -229.112,A -90.000,B 90.000,C 0.000} C_DIS
LIN {X 107.869,Y -7.144,Z -232.754,A -90.000,B 90.000,C 0.000} C_DIS
LIN {X 106.741,Y -7.144,Z -236.378,A -90.000,B 90.000,C 0.000} C_DIS
LIN {X 105.550,Y -7.144,Z -239.980,A -90.000,B 90.000,C 0.000} C_DIS
LIN {X 104.295,Y -7.144,Z -243.561,A -90.000,B 90.000,C 0.000} C_DIS
LIN {X 145.015,Y -7.144,Z -243.561,A -90.000,B 90.000,C 0.000} C_DIS
LIN {X 145.015,Y -19.644,Z -243.561,A -90.000,B 90.000,C 0.000} C_DIS
LIN {X 145.015,Y -32.144,Z -243.561,A -90.000,B 90.000,C 0.000} C_DIS
LIN {X 145.015,Y -57.084,Z -243.561,A -90.000,B 90.000,C 0.000} C_DIS
LIN {X -144.015,Y -57.084,Z -242.561,A -90.000,B 90.000,C 0.000} C_DIS
LIN {X -144.015,Y -25.000,Z -242.561,A -90.000,B 90.000,C 0.000} C_DIS
LIN {X -144.015,Y -12.500,Z -242.561,A -90.000,B 90.000,C 0.000} C_DIS
LIN {X -144.015,Y 0.000,Z -242.561,A -90.000,B 90.000,C 0.000} C_DIS
LIN {X -141.861,Y 0.000,Z -242.561,A -90.000,B 90.000,C 0.000} C_DIS
LIN {X -141.450,Y 0.000,Z -241.919,A -90.000,B 90.000,C 0.000} C_DIS
LIN {X -141.001,Y 0.000,Z -241.303,A -90.000,B 90.000,C 0.000} C_DIS
LIN {X -140.515,Y 0.000,Z -240.715,A -90.000,B 90.000,C 0.000} C_DIS
LIN {X -139.994,Y 0.000,Z -240.158,A -90.000,B 90.000,C 0.000} C_DIS
LIN {X -139.440,Y 0.000,Z -239.634,A -90.000,B 90.000,C 0.000} C_DIS
LIN {X -138.855,Y 0.000,Z -239.145,A -90.000,B 90.000,C 0.000} C_DIS
LIN {X -136.796,Y 0.000,Z -237.735,A -90.000,B 90.000,C 0.000} C_DIS
LIN {X -134.714,Y 0.000,Z -236.357,A -90.000,B 90.000,C 0.000} C_DIS
LIN {X -132.612,Y 0.000,Z -235.012,A -90.000,B 90.000,C 0.000} C_DIS
LIN {X -144.015,Y 0.000,Z -235.012,A -90.000,B 90.000,C 0.000} C_DIS
LIN {X -144.015,Y 0.000,Z -227.464,A -90.000,B 90.000,C 0.000} C_DIS
LIN {X -132.537,Y 0.000,Z -227.464,A -90.000,B 90.000,C 0.000} C_DIS
LIN {X -132.537,Y 0.000,Z -219.915,A -90.000,B 90.000,C 0.000} C_DIS
LIN {X -144.015,Y 0.000,Z -219.915,A -90.000,B 90.000,C 0.000} C_DIS
LIN {X -144.015,Y 0.000,Z -212.366,A -90.000,B 90.000,C 0.000} C_DIS
LIN {X -132.537,Y 0.000,Z -212.366,A -90.000,B 90.000,C 0.000} C_DIS
LIN {X -132.537,Y 0.000,Z -204.817,A -90.000,B 90.000,C 0.000} C_DIS
LIN {X -144.015,Y 0.000,Z -204.817,A -90.000,B 90.000,C 0.000} C_DIS
LIN {X -144.015,Y 0.000,Z -197.269,A -90.000,B 90.000,C 0.000} C_DIS
LIN {X -132.537,Y 0.000,Z -197.269,A -90.000,B 90.000,C 0.000} C_DIS
LIN {X -132.537,Y 0.000,Z -189.720,A -90.000,B 90.000,C 0.000} C_DIS
LIN {X -144.015,Y 0.000,Z -189.720,A -90.000,B 90.000,C 0.000} C_DIS
LIN {X -144.015,Y 0.000,Z -182.171,A -90.000,B 90.000,C 0.000} C_DIS
LIN {X -132.537,Y 0.000,Z -182.171,A -90.000,B 90.000,C 0.000} C_DIS
LIN {X -132.537,Y 0.000,Z -174.622,A -90.000,B 90.000,C 0.000} C_DIS
LIN {X -144.015,Y 0.000,Z -174.622,A -90.000,B 90.000,C 0.000} C_DIS
LIN {X -144.015,Y 0.000,Z -167.073,A -90.000,B 90.000,C 0.000} C_DIS
LIN {X -132.537,Y 0.000,Z -167.073,A -90.000,B 90.000,C 0.000} C_DIS
LIN {X -132.537,Y 0.000,Z -159.525,A -90.000,B 90.000,C 0.000} C_DIS
LIN {X -144.015,Y 0.000,Z -159.525,A -90.000,B 90.000,C 0.000} C_DIS
LIN {X -144.015,Y 0.000,Z -151.976,A -90.000,B 90.000,C 0.000} C_DIS
LIN {X -132.537,Y 0.000,Z -151.976,A -90.000,B 90.000,C 0.000} C_DIS
LIN {X -132.537,Y 0.000,Z -144.427,A -90.000,B 90.000,C 0.000} C_DIS
LIN {X -144.015,Y 0.000,Z -144.427,A -90.000,B 90.000,C 0.000} C_DIS
LIN {X -144.015,Y 0.000,Z -136.878,A -90.000,B 90.000,C 0.000} C_DIS
LIN {X -132.537,Y 0.000,Z -136.878,A -90.000,B 90.000,C 0.000} C_DIS
LIN {X -132.537,Y 0.000,Z -129.329,A -90.000,B 90.000,C 0.000} C_DIS
LIN {X -144.015,Y 0.000,Z -129.329,A -90.000,B 90.000,C 0.000} C_DIS
LIN {X -144.015,Y 0.000,Z -121.781,A -90.000,B 90.000,C 0.000} C_DIS
LIN {X -132.537,Y 0.000,Z -121.781,A -90.000,B 90.000,C 0.000} C_DIS
LIN {X -132.537,Y 0.000,Z -114.232,A -90.000,B 90.000,C 0.000} C_DIS
LIN {X -144.015,Y 0.000,Z -114.232,A -90.000,B 90.000,C 0.000} C_DIS
LIN {X -144.015,Y 0.000,Z -106.683,A -90.000,B 90.000,C 0.000} C_DIS
LIN {X -132.537,Y 0.000,Z -106.683,A -90.000,B 90.000,C 0.000} C_DIS
LIN {X -132.537,Y 0.000,Z -99.134,A -90.000,B 90.000,C 0.000} C_DIS
LIN {X -144.015,Y 0.000,Z -99.134,A -90.000,B 90.000,C 0.000} C_DIS
LIN {X -144.015,Y 0.000,Z -91.586,A -90.000,B 90.000,C 0.000} C_DIS
LIN {X -132.537,Y 0.000,Z -91.586,A -90.000,B 90.000,C 0.000} C_DIS
LIN {X -132.537,Y 0.000,Z -84.037,A -90.000,B 90.000,C 0.000} C_DIS
LIN {X -144.015,Y 0.000,Z -84.037,A -90.000,B 90.000,C 0.000} C_DIS
LIN {X -144.015,Y 0.000,Z -76.488,A -90.000,B 90.000,C 0.000} C_DIS
LIN {X -132.537,Y 0.000,Z -76.488,A -90.000,B 90.000,C 0.000} C_DIS
LIN {X -132.537,Y 0.000,Z -68.939,A -90.000,B 90.000,C 0.000} C_DIS
LIN {X -144.015,Y 0.000,Z -68.939,A -90.000,B 90.000,C 0.000} C_DIS
LIN {X -144.015,Y 0.000,Z -61.390,A -90.000,B 90.000,C 0.000} C_DIS
LIN {X -132.537,Y 0.000,Z -61.390,A -90.000,B 90.000,C 0.000} C_DIS
LIN {X -132.537,Y 0.000,Z -53.842,A -90.000,B 90.000,C 0.000} C_DIS
LIN {X -144.015,Y 0.000,Z -53.842,A -90.000,B 90.000,C 0.000} C_DIS
LIN {X -144.015,Y 0.000,Z -46.293,A -90.000,B 90.000,C 0.000} C_DIS
LIN {X -132.537,Y 0.000,Z -46.293,A -90.000,B 90.000,C 0.000} C_DIS
LIN {X -132.537,Y 0.000,Z -38.744,A -90.000,B 90.000,C 0.000} C_DIS
LIN {X -144.015,Y 0.000,Z -38.744,A -90.000,B 90.000,C 0.000} C_DIS
LIN {X -144.015,Y 0.000,Z -31.195,A -90.000,B 90.000,C 0.000} C_DIS
LIN {X -132.537,Y 0.000,Z -31.195,A -90.000,B 90.000,C 0.000} C_DIS
LIN {X -132.537,Y 0.000,Z -23.646,A -90.000,B 90.000,C 0.000} C_DIS
LIN {X -144.015,Y 0.000,Z -23.646,A -90.000,B 90.000,C 0.000} C_DIS
LIN {X -144.015,Y 0.000,Z -16.098,A -90.000,B 90.000,C 0.000} C_DIS
LIN {X -132.537,Y 0.000,Z -16.098,A -90.000,B 90.000,C 0.000} C_DIS
LIN {X -132.537,Y 0.000,Z -8.549,A -90.000,B 90.000,C 0.000} C_DIS
LIN {X -144.015,Y 0.000,Z -8.549,A -90.000,B 90.000,C 0.000} C_DIS
LIN {X -144.015,Y 0.000,Z -1.000,A -90.000,B 90.000,C 0.000} C_DIS
LIN {X -132.537,Y 0.000,Z -1.000,A -90.000,B 90.000,C 0.000} C_DIS
LIN {X -131.537,Y 0.000,Z -0.237,A -90.000,B 90.000,C 0.000} C_DIS
LIN {X -131.527,Y 0.000,Z 0.000,A -90.000,B 90.000,C 0.000} C_DIS
LIN {X -145.015,Y 0.000,Z 0.000,A -90.000,B 90.000,C 0.000} C_DIS
LIN {X -145.015,Y 0.000,Z -243.561,A -90.000,B 90.000,C 0.000} C_DIS
LIN {X -141.266,Y 0.000,Z -243.561,A -90.000,B 90.000,C 0.000} C_DIS
LIN {X -141.189,Y 0.000,Z -243.399,A -90.000,B 90.000,C 0.000} C_DIS
LIN {X -140.799,Y 0.000,Z -242.748,A -90.000,B 90.000,C 0.000} C_DIS
LIN {X -140.367,Y 0.000,Z -242.123,A -90.000,B 90.000,C 0.000} C_DIS
LIN {X -139.895,Y 0.000,Z -241.529,A -90.000,B 90.000,C 0.000} C_DIS
LIN {X -139.385,Y 0.000,Z -240.967,A -90.000,B 90.000,C 0.000} C_DIS
LIN {X -138.839,Y 0.000,Z -240.440,A -90.000,B 90.000,C 0.000} C_DIS
LIN {X -138.260,Y 0.000,Z -239.949,A -90.000,B 90.000,C 0.000} C_DIS
LIN {X -136.044,Y 0.000,Z -238.435,A -90.000,B 90.000,C 0.000} C_DIS
LIN {X -133.803,Y 0.000,Z -236.958,A -90.000,B 90.000,C 0.000} C_DIS
LIN {X -131.537,Y 0.000,Z -235.520,A -90.000,B 90.000,C 0.000} C_DIS
LIN {X -131.537,Y 0.000,Z -0.237,A -90.000,B 90.000,C 0.000} C_DIS
LIN {X -131.537,Y -12.500,Z -0.237,A -90.000,B 90.000,C 0.000} C_DIS
LIN {X -131.537,Y -75.000,Z -0.237,A -90.000,B 90.000,C 0.000} C_DIS
LIN {X 132.540,Y -75.000,Z -242.561,A -90.000,B 90.000,C 0.000} C_DIS
LIN {X 132.540,Y -12.500,Z -242.561,A -90.000,B 90.000,C 0.000} C_DIS
LIN {X 132.540,Y 0.000,Z -242.561,A -90.000,B 90.000,C 0.000} C_DIS
LIN {X 144.015,Y 0.000,Z -242.561,A -90.000,B 90.000,C 0.000} C_DIS
LIN {X 144.015,Y 0.000,Z -235.012,A -90.000,B 90.000,C 0.000} C_DIS
LIN {X 132.540,Y 0.000,Z -235.012,A -90.000,B 90.000,C 0.000} C_DIS
LIN {X 132.540,Y 0.000,Z -227.464,A -90.000,B 90.000,C 0.000} C_DIS
LIN {X 144.015,Y 0.000,Z -227.464,A -90.000,B 90.000,C 0.000} C_DIS
LIN {X 144.015,Y 0.000,Z -219.915,A -90.000,B 90.000,C 0.000} C_DIS
LIN {X 132.540,Y 0.000,Z -219.915,A -90.000,B 90.000,C 0.000} C_DIS
LIN {X 132.540,Y 0.000,Z -212.366,A -90.000,B 90.000,C 0.000} C_DIS
LIN {X 144.015,Y 0.000,Z -212.366,A -90.000,B 90.000,C 0.000} C_DIS
LIN {X 144.015,Y 0.000,Z -204.817,A -90.000,B 90.000,C 0.000} C_DIS
LIN {X 132.540,Y 0.000,Z -204.817,A -90.000,B 90.000,C 0.000} C_DIS
LIN {X 132.540,Y 0.000,Z -197.269,A -90.000,B 90.000,C 0.000} C_DIS
LIN {X 144.015,Y 0.000,Z -197.269,A -90.000,B 90.000,C 0.000} C_DIS
LIN {X 144.015,Y 0.000,Z -189.720,A -90.000,B 90.000,C 0.000} C_DIS
LIN {X 132.540,Y 0.000,Z -189.720,A -90.000,B 90.000,C 0.000} C_DIS
LIN {X 132.540,Y 0.000,Z -182.171,A -90.000,B 90.000,C 0.000} C_DIS
LIN {X 144.015,Y 0.000,Z -182.171,A -90.000,B 90.000,C 0.000} C_DIS
LIN {X 144.015,Y 0.000,Z -174.622,A -90.000,B 90.000,C 0.000} C_DIS
LIN {X 132.540,Y 0.000,Z -174.622,A -90.000,B 90.000,C 0.000} C_DIS
LIN {X 132.540,Y 0.000,Z -167.073,A -90.000,B 90.000,C 0.000} C_DIS
LIN {X 144.015,Y 0.000,Z -167.073,A -90.000,B 90.000,C 0.000} C_DIS
LIN {X 144.015,Y 0.000,Z -159.525,A -90.000,B 90.000,C 0.000} C_DIS
LIN {X 132.540,Y 0.000,Z -159.525,A -90.000,B 90.000,C 0.000} C_DIS
LIN {X 132.540,Y 0.000,Z -151.976,A -90.000,B 90.000,C 0.000} C_DIS
LIN {X 144.015,Y 0.000,Z -151.976,A -90.000,B 90.000,C 0.000} C_DIS
LIN {X 144.015,Y 0.000,Z -144.427,A -90.000,B 90.000,C 0.000} C_DIS
LIN {X 132.540,Y 0.000,Z -144.427,A -90.000,B 90.000,C 0.000} C_DIS
LIN {X 132.540,Y 0.000,Z -136.878,A -90.000,B 90.000,C 0.000} C_DIS
LIN {X 144.015,Y 0.000,Z -136.878,A -90.000,B 90.000,C 0.000} C_DIS
LIN {X 144.015,Y 0.000,Z -129.329,A -90.000,B 90.000,C 0.000} C_DIS
LIN {X 132.540,Y 0.000,Z -129.329,A -90.000,B 90.000,C 0.000} C_DIS
LIN {X 132.540,Y 0.000,Z -121.781,A -90.000,B 90.000,C 0.000} C_DIS
LIN {X 144.015,Y 0.000,Z -121.781,A -90.000,B 90.000,C 0.000} C_DIS
LIN {X 144.015,Y 0.000,Z -114.232,A -90.000,B 90.000,C 0.000} C_DIS
LIN {X 132.540,Y 0.000,Z -114.232,A -90.000,B 90.000,C 0.000} C_DIS
LIN {X 132.540,Y 0.000,Z -106.683,A -90.000,B 90.000,C 0.000} C_DIS
LIN {X 144.015,Y 0.000,Z -106.683,A -90.000,B 90.000,C 0.000} C_DIS
LIN {X 144.015,Y 0.000,Z -99.134,A -90.000,B 90.000,C 0.000} C_DIS
LIN {X 132.540,Y 0.000,Z -99.134,A -90.000,B 90.000,C 0.000} C_DIS
LIN {X 132.540,Y 0.000,Z -91.586,A -90.000,B 90.000,C 0.000} C_DIS
LIN {X 144.015,Y 0.000,Z -91.586,A -90.000,B 90.000,C 0.000} C_DIS
LIN {X 144.015,Y 0.000,Z -84.037,A -90.000,B 90.000,C 0.000} C_DIS
LIN {X 132.540,Y 0.000,Z -84.037,A -90.000,B 90.000,C 0.000} C_DIS
LIN {X 132.540,Y 0.000,Z -76.488,A -90.000,B 90.000,C 0.000} C_DIS
LIN {X 144.015,Y 0.000,Z -76.488,A -90.000,B 90.000,C 0.000} C_DIS
LIN {X 144.015,Y 0.000,Z -68.939,A -90.000,B 90.000,C 0.000} C_DIS
LIN {X 132.540,Y 0.000,Z -68.939,A -90.000,B 90.000,C 0.000} C_DIS
LIN {X 132.540,Y 0.000,Z -61.390,A -90.000,B 90.000,C 0.000} C_DIS
LIN {X 144.015,Y 0.000,Z -61.390,A -90.000,B 90.000,C 0.000} C_DIS
LIN {X 144.015,Y 0.000,Z -53.842,A -90.000,B 90.000,C 0.000} C_DIS
LIN {X 132.540,Y 0.000,Z -53.842,A -90.000,B 90.000,C 0.000} C_DIS
LIN {X 132.540,Y 0.000,Z -46.293,A -90.000,B 90.000,C 0.000} C_DIS
LIN {X 144.015,Y 0.000,Z -46.293,A -90.000,B 90.000,C 0.000} C_DIS
LIN {X 144.015,Y 0.000,Z -38.744,A -90.000,B 90.000,C 0.000} C_DIS
LIN {X 132.540,Y 0.000,Z -38.744,A -90.000,B 90.000,C 0.000} C_DIS
LIN {X 132.540,Y 0.000,Z -31.195,A -90.000,B 90.000,C 0.000} C_DIS
LIN {X 144.015,Y 0.000,Z -31.195,A -90.000,B 90.000,C 0.000} C_DIS
LIN {X 144.015,Y 0.000,Z -23.646,A -90.000,B 90.000,C 0.000} C_DIS
LIN {X 132.540,Y 0.000,Z -23.646,A -90.000,B 90.000,C 0.000} C_DIS
LIN {X 132.540,Y 0.000,Z -16.098,A -90.000,B 90.000,C 0.000} C_DIS
LIN {X 144.015,Y 0.000,Z -16.098,A -90.000,B 90.000,C 0.000} C_DIS
LIN {X 144.015,Y 0.000,Z -8.549,A -90.000,B 90.000,C 0.000} C_DIS
LIN {X 132.540,Y 0.000,Z -8.549,A -90.000,B 90.000,C 0.000} C_DIS
LIN {X 132.540,Y 0.000,Z -1.000,A -90.000,B 90.000,C 0.000} C_DIS
LIN {X 144.015,Y 0.000,Z -1.000,A -90.000,B 90.000,C 0.000} C_DIS
LIN {X 145.015,Y 0.000,Z 0.000,A -90.000,B 90.000,C 0.000} C_DIS
LIN {X 131.540,Y 0.000,Z 0.000,A -90.000,B 90.000,C 0.000} C_DIS
LIN {X 131.540,Y 0.000,Z -243.561,A -90.000,B 90.000,C 0.000} C_DIS
LIN {X 145.015,Y 0.000,Z -243.561,A -90.000,B 90.000,C 0.000} C_DIS
LIN {X 145.015,Y 0.000,Z 0.000,A -90.000,B 90.000,C 0.000} C_DIS
LIN {X 145.015,Y -5.000,Z 0.000,A -90.000,B 90.000,C 0.000} C_DIS
LIN {X 145.015,Y -75.000,Z 0.000,A -90.000,B 90.000,C 0.000} C_DIS

END
